(* Schneider Machine Expert - Basic project Redundant_Motors_TM221CE16T, file version 3.0.0.0 *)
(* ProjectInformations: Name=New project *)

HARDWARE
  Cpu 0: TM221CE16T
  EthernetConfiguration: NetworkName=M221, IpAllocationMode=FixedAddress, IpAddress=0.0.0.0, SubnetMask=0.0.0.0
  SerialLineConfiguration: Baud=Baud19200, Parity=ParityEven, DataBits=DataBits8, StopBits=StopBits1, PhysicalMedium=PhysicalMediumRs485, TransmissionMode=TransmissionModeModbusRtu, SlaveId=1, Addressing=SlaveAddressing
  MastTask: UsePeriodScanMode=false, PeriodScan=100
  FastTask: Period=255
  CpuBehavior: StartingMode=StartAsPreviousState, AutoSaveRamOnEeprom=true, WatchdogPeriod=250

SYMBOLS  (address, symbol, comment, settings)
  %M0       SYSTEM_READY
  %S0       SB_COLDSTART  "Indicates or executes a cold start (data initialized to default values)"
  %S1       SB_WARMSTART  "Indicates there was a warm start with data backup"
  %TM0        [Preset=3, Base=OneSecond]
  %TM1        [Preset=5, Base=OneSecond]
  %TM2        [Preset=5, Base=OneSecond]
  %I0.0     EMERGENCY_PB

POU New POU
  (* SectionNumber=0 *)

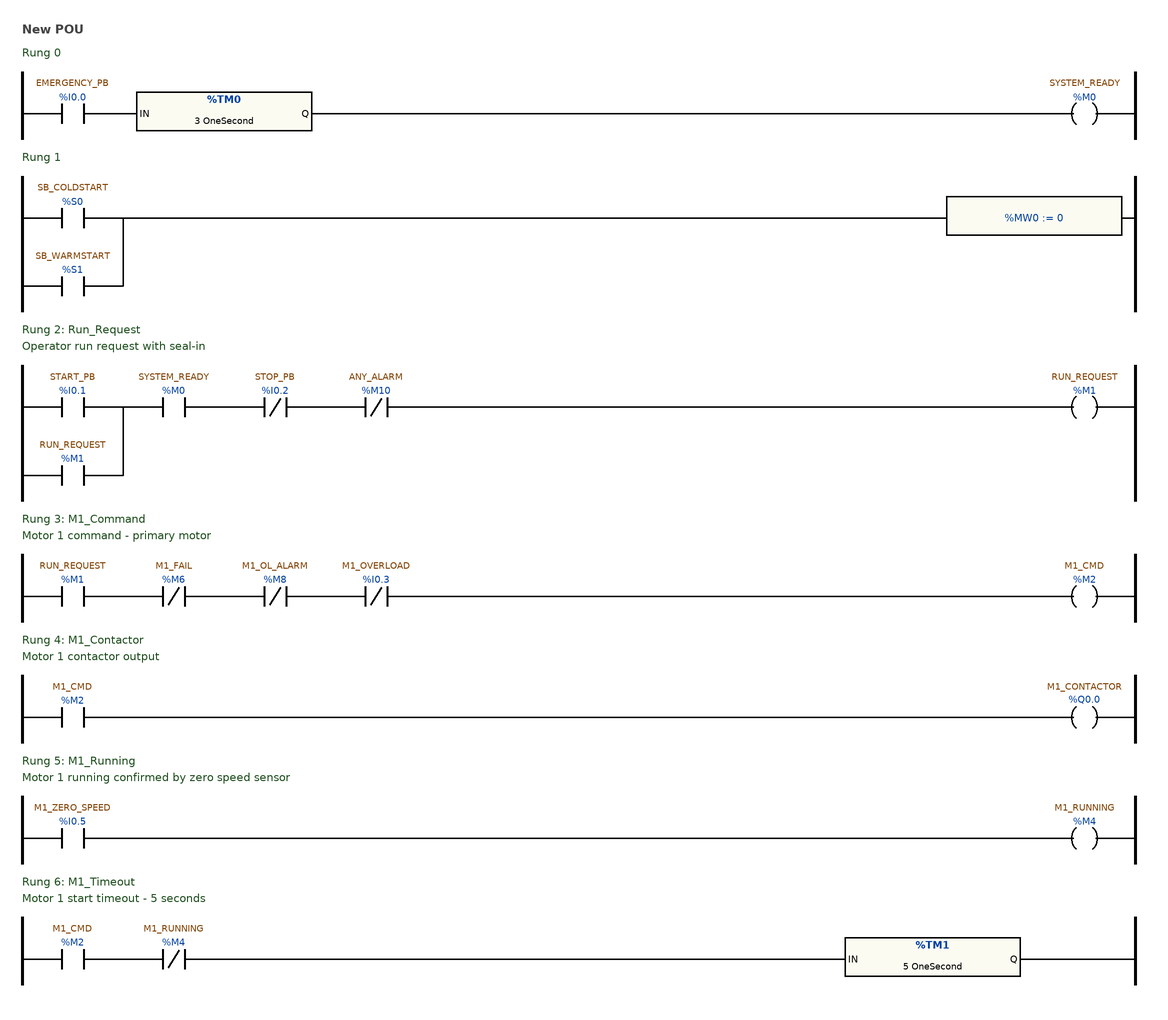

// Rung 0
  BLK %TM0
  LD %I0.0                (* EMERGENCY_PB *)
  IN
  OUT_BLK
  LD Q
  ST %M0                  (* SYSTEM_READY *)
  END_BLK
  // as ST:
  //   %TM0(IN := EMERGENCY_PB);
  //   SYSTEM_READY := %TM0.Q;

// Rung 1
  LD %S0                  (* SB_COLDSTART *)
  OR %S1                  (* SB_WARMSTART *)
  [ %MW0 := 0 ]
  // as ST:
  //   IF SB_COLDSTART OR SB_WARMSTART THEN %MW0 := 0; END_IF;

// Rung 2: Run_Request
// Operator run request with seal-in
  LD %I0.1
  OR %M1
  AND %M0                 (* SYSTEM_READY *)
  ANDN %I0.2
  ANDN %M10
  ST %M1
  // %I0.1: Start Button
  // %M0: System Ready
  // %I0.2: Stop NC
  // %M10: No Alarm
  // %M1: Run Request
  // %M1: Seal-in
  // as ST:
  //   %M1 := (%I0.1 OR %M1) AND SYSTEM_READY AND NOT %I0.2 AND NOT %M10;

// Rung 3: M1_Command
// Motor 1 command - primary motor
  LD %M1
  ANDN %M6
  ANDN %M8
  ANDN %I0.3
  ST %M2
  // %M1: Run Req
  // %M6: M1 OK
  // %M8: No OL
  // %I0.3: OL OK
  // %M2: M1 Cmd
  // as ST:
  //   %M2 := %M1 AND NOT %M6 AND NOT %M8 AND NOT %I0.3;

// Rung 4: M1_Contactor
// Motor 1 contactor output
  LD %M2
  ST %Q0.0
  // %M2: M1 Cmd
  // %Q0.0: M1 Cont
  // as ST:
  //   %Q0.0 := %M2;

// Rung 5: M1_Running
// Motor 1 running confirmed by zero speed sensor
  LD %I0.5
  ST %M4
  // %I0.5: M1 Speed
  // %M4: M1 Run
  // as ST:
  //   %M4 := %I0.5;

// Rung 6: M1_Timeout
// Motor 1 start timeout - 5 seconds
  BLK %TM1
  LD %M2
  ANDN %M4
  IN
  OUT_BLK
  END_BLK
  // %M2: M1 Cmd
  // %M4: Not Run
  // %TM1: 5s
  // as ST:
  //   %TM1(IN := %M2 AND NOT %M4);

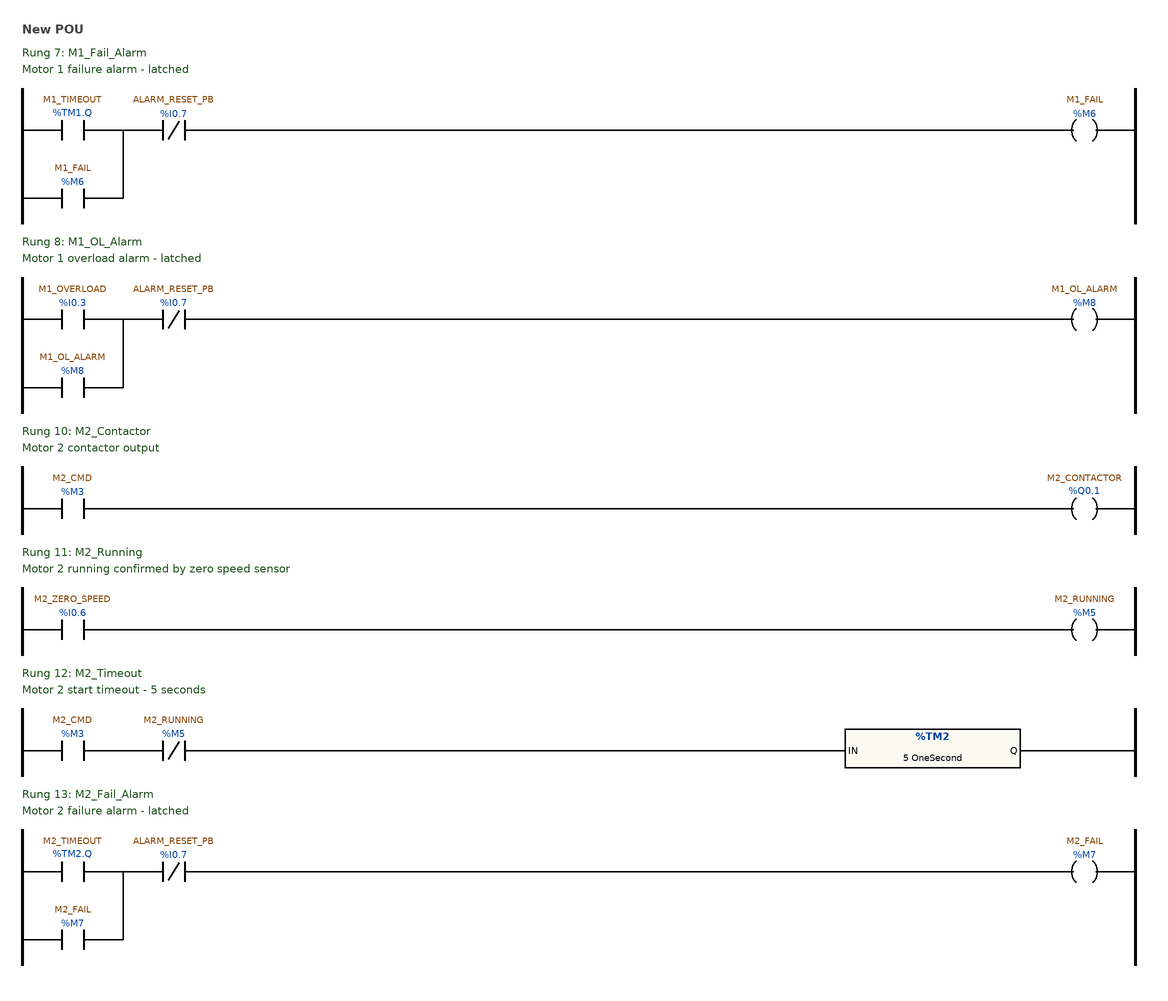

// Rung 7: M1_Fail_Alarm
// Motor 1 failure alarm - latched
  LD %TM1.Q
  OR %M6
  ANDN %I0.7
  ST %M6
  // %TM1.Q: Timeout
  // %I0.7: No Reset
  // %M6: M1 Fail
  // %M6: Latch
  // as ST:
  //   %M6 := (%TM1.Q OR %M6) AND NOT %I0.7;

// Rung 8: M1_OL_Alarm
// Motor 1 overload alarm - latched
  LD %I0.3
  OR %M8
  ANDN %I0.7
  ST %M8
  // %I0.3: M1 OL
  // %I0.7: No Reset
  // %M8: M1 OL Alm
  // %M8: Latch
  // as ST:
  //   %M8 := (%I0.3 OR %M8) AND NOT %I0.7;

// Rung 9: M2_Command
// Motor 2 backup - auto-starts when M1 fails or overloads
  LD %M1
  AND( %M6
  OR %M8
  )
  ANDN %M7
  ANDN %M9
  ANDN %I0.4
  ST %M3
  // %M1: Run Req
  // %M6: M1 Fail
  // %M7: M2 OK
  // %M9: No OL
  // %I0.4: OL OK
  // %M3: M2 Cmd
  // %M8: M1 OL
  // as ST:
  //   %M3 := %M1 AND (%M6 OR %M8) AND NOT %M7 AND NOT %M9 AND NOT %I0.4;
  (* the ladder stored for this rung does not match its IL; not drawn *)

// Rung 10: M2_Contactor
// Motor 2 contactor output
  LD %M3
  ST %Q0.1
  // %M3: M2 Cmd
  // %Q0.1: M2 Cont
  // as ST:
  //   %Q0.1 := %M3;

// Rung 11: M2_Running
// Motor 2 running confirmed by zero speed sensor
  LD %I0.6
  ST %M5
  // %I0.6: M2 Speed
  // %M5: M2 Run
  // as ST:
  //   %M5 := %I0.6;

// Rung 12: M2_Timeout
// Motor 2 start timeout - 5 seconds
  BLK %TM2
  LD %M3
  ANDN %M5
  IN
  OUT_BLK
  END_BLK
  // %M3: M2 Cmd
  // %M5: Not Run
  // %TM2: 5s
  // as ST:
  //   %TM2(IN := %M3 AND NOT %M5);

// Rung 13: M2_Fail_Alarm
// Motor 2 failure alarm - latched
  LD %TM2.Q
  OR %M7
  ANDN %I0.7
  ST %M7
  // %TM2.Q: Timeout
  // %I0.7: No Reset
  // %M7: M2 Fail
  // %M7: Latch
  // as ST:
  //   %M7 := (%TM2.Q OR %M7) AND NOT %I0.7;

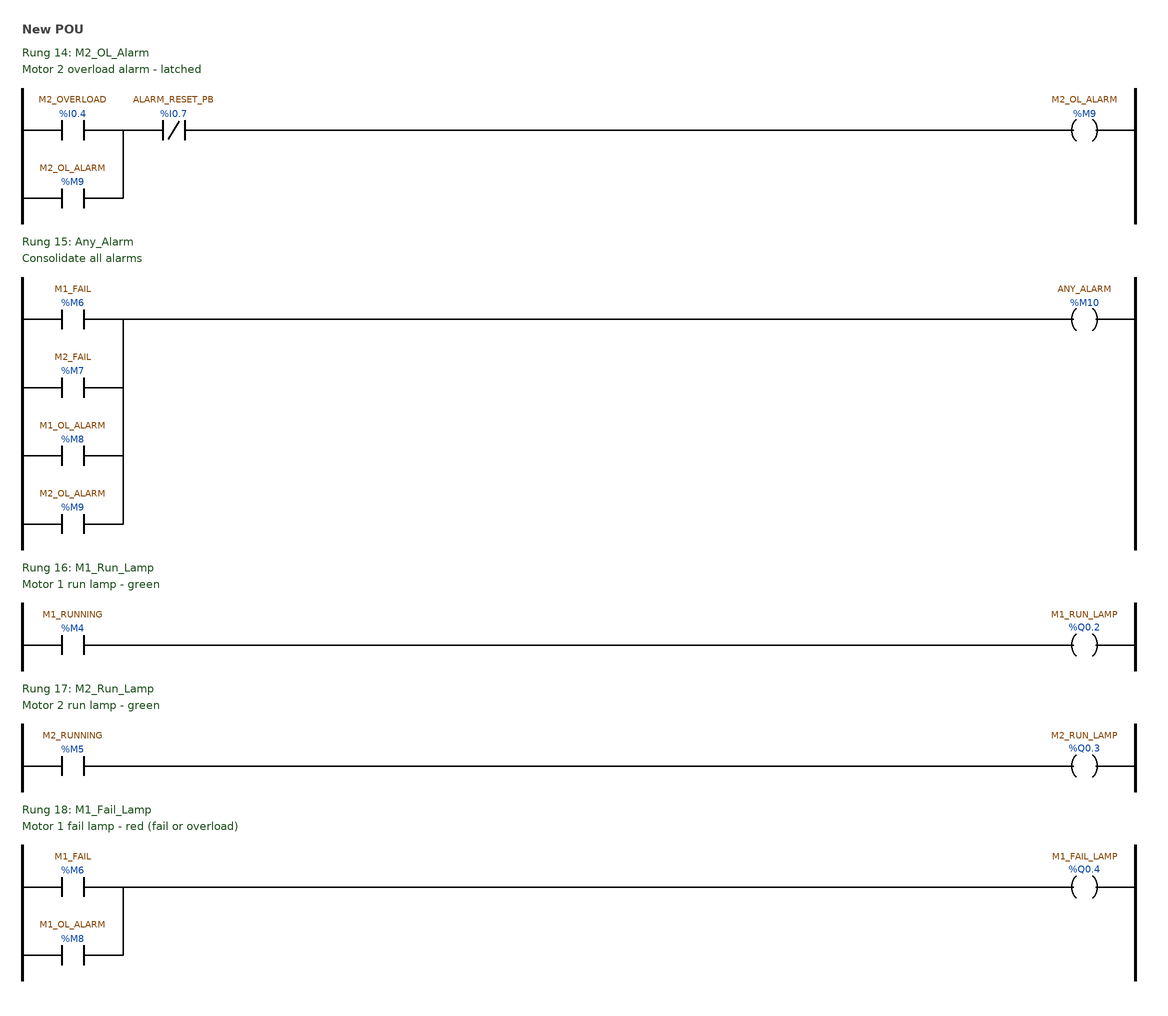

// Rung 14: M2_OL_Alarm
// Motor 2 overload alarm - latched
  LD %I0.4
  OR %M9
  ANDN %I0.7
  ST %M9
  // %I0.4: M2 OL
  // %I0.7: No Reset
  // %M9: M2 OL Alm
  // %M9: Latch
  // as ST:
  //   %M9 := (%I0.4 OR %M9) AND NOT %I0.7;

// Rung 15: Any_Alarm
// Consolidate all alarms
  LD %M6
  OR %M7
  OR %M8
  OR %M9
  ST %M10
  // %M6: M1 Fail
  // %M10: Any Alm
  // %M7: M2 Fail
  // %M8: M1 OL
  // %M9: M2 OL
  // as ST:
  //   %M10 := %M6 OR %M7 OR %M8 OR %M9;

// Rung 16: M1_Run_Lamp
// Motor 1 run lamp - green
  LD %M4
  ST %Q0.2
  // %M4: M1 Run
  // %Q0.2: M1 Lamp
  // as ST:
  //   %Q0.2 := %M4;

// Rung 17: M2_Run_Lamp
// Motor 2 run lamp - green
  LD %M5
  ST %Q0.3
  // %M5: M2 Run
  // %Q0.3: M2 Lamp
  // as ST:
  //   %Q0.3 := %M5;

// Rung 18: M1_Fail_Lamp
// Motor 1 fail lamp - red (fail or overload)
  LD %M6
  OR %M8
  ST %Q0.4
  // %M6: M1 Fail
  // %Q0.4: M1 Fail Lp
  // %M8: M1 OL
  // as ST:
  //   %Q0.4 := %M6 OR %M8;

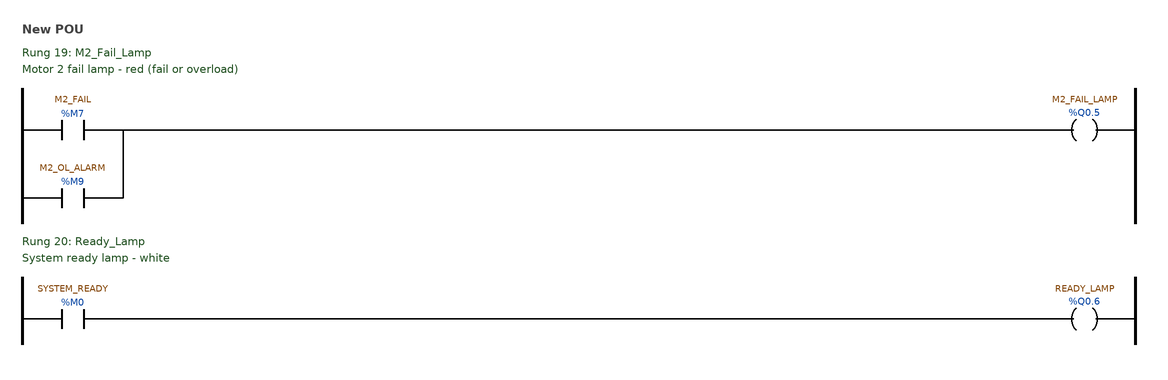

// Rung 19: M2_Fail_Lamp
// Motor 2 fail lamp - red (fail or overload)
  LD %M7
  OR %M9
  ST %Q0.5
  // %M7: M2 Fail
  // %Q0.5: M2 Fail Lp
  // %M9: M2 OL
  // as ST:
  //   %Q0.5 := %M7 OR %M9;

// Rung 20: Ready_Lamp
// System ready lamp - white
  LD %M0                  (* SYSTEM_READY *)
  ST %Q0.6
  // %M0: Ready
  // %Q0.6: Ready Lp
  // as ST:
  //   %Q0.6 := SYSTEM_READY;
